(* IEC 61131-3 sources: learning-path/06_oop_in_st/exercises/1_interfaces/src, 2 files *)

(* ---- ItfValve.st ---- *)
//File to create the interface to implement the class valve
//File to create the interface to implement the class tank
NAMESPACE FluidHandlingClass

    INTERFACE ItfValve
    END_INTERFACE

END_NAMESPACE

(* ---- TankBase.st ---- *)
//Use the same namespace than the TYPE for the Valves state

NAMESPACE FluidHandlingClass

    CLASS TankBase
        VAR PRIVATE
            inletValve: ValveBase;
            outletValve: ValveBase;
        END_VAR

        METHOD PUBLIC Fill
            inletValve.Open();
            outletValve.Close();
        END_METHOD

        METHOD PUBLIC Flush
            inletValve.Open();
            outletValve.Open();
        END_METHOD

        METHOD PUBLIC Close
            inletValve.Close();
            outletValve.Close();
        END_METHOD

        METHOD PUBLIC Emptying
            this.Close();
            outletValve.Open();
        END_METHOD
    END_CLASS

END_NAMESPACE
